{attribute 'GeneratedUsingTerminal: EK1122-0000-0018'}
{attribute addProperty BoxType "EK1122-0000-0018"}
{attribute addProperty Id "Beckhoff_EL47xxsub_EK1100EK1100_1FC0878B2"}
{attribute addProperty CRC "3661231638"}
{attribute addProperty Size "2"}
TYPE Beckhoff_EL47xxEK1122_DA39F616 EXTENDS EK1122_1FC0878B :
STRUCT
	{attribute addProperty Name "Beckhoff_EL47xxsub_EK1100"}
	{attribute addProperty PreviousPort "Beckhoff EL47xxEK1122 : D"}
	Beckhoff_EL47xxsub_EK1100 : EK1100_1FC0878B;
END_STRUCT
END_TYPE

(* stored: Version 1.2.0.0, ProductVersion 3.1.4024.9
   DUT Beckhoff_EL47xxEK1122_DA39F616: Id {a14c6743-7251-4db7-b0c0-0701b30b8482} *)
